# B&R Automation Studio project prac1
Automation Studio 4.12.10.39

## Configuration Config1

CPU PC_any, AutomationRuntime J4.93, Build 4.1.2, Vc V4.73.2

### Task classes (Cpu.sw)
```
Cyclic#1 (cycle 10000 us):
  Program <- Program.prg
Cyclic#4:
  Program1 <- Program1.prg
Binaries: udbdef, FWRules, TCData, sysconf, Role, User, iomap, ashwd, asfw, arconfig, ashwac
Libraries: Library
```

### Hardware
```
PC : PC_any v1.1.1.0 (OrderNumber=PC)
  ConfigurationID = prac1_Config1
  Cyclic1Duration = 10000
  Cyclic2Duration = 100000
  Cyclic3Duration = 300000
  Cyclic3Tolerance = 9900000
  FileDevice1
  FileDeviceName1 = USER
  FileDevicePath1 = USER_PATH
```

- Physical/Config1/PC/IoMap.iom: same as Physical/Config1/PC/Cpu.per
- Physical/Config1/PC/PvMap.vvm: same as Physical/Config1/PC/Cpu.per
## Logical view

Binary libraries used (declarations not repeated): operator, runtime, astime, AsIecCon

### Global.var - Global variables
```iecst
VAR
	Enable : BOOL := TRUE;
	Speed : INT;
END_VAR
```


### Program Logical/Program (ANSIC)

#### Main.c - Init, cyclic, exit code
```c
#include <bur/plctypes.h>

#ifdef _DEFAULT_INCLUDES
	#include <AsDefault.h>
#endif

void _INIT ProgramInit(void)
{
	REAL Tj = 1;
	REAL D_T = 0.01;

	fb_motor.Tm = 0.1;
	fb_motor.ke = 0.24;
	fb_motor.dt = D_T;
	fb_motor.integrator.dt = D_T;

	fb_regulator.k_p = fb_motor.ke * fb_motor.Tm / Tj;
	fb_regulator.k_i = fb_motor.ke / Tj;
	fb_regulator.dt  = D_T;
	fb_regulator.max_abs_value = 24.0;
	fb_regulator.integrator.dt = D_T;

	fb_motor_2.Tm = 0.1;
	fb_motor_2.ke = 0.24;
	fb_motor_2.dt = D_T;
	fb_motor_2.integrator.dt = D_T;

}

void _CYCLIC ProgramCyclic(void)
{

	if (Enable)
	{
		fb_regulator.e = Speed - fb_motor.w;
		FB_regulator(&fb_regulator);

		fb_motor.u = fb_regulator.u;
		FB_motor(&fb_motor);

		fb_motor_2.u = Speed * fb_motor_2.ke;
		FB_motor(&fb_motor_2);
	}
	else
	{
		fb_regulator.u = 0.0;
		fb_regulator.iyOld = 0.0;
		fb_regulator.integrator.out = 0.0;

		fb_motor.u = 0.0;
		FB_motor(&fb_motor);

		fb_motor_2.u = 0;
		FB_motor(&fb_motor_2);
	}
}
void _EXIT ProgramExit(void)
{

}
```

#### Variables.var - Local variables
```iecst
VAR
	fb_regulator : FB_regulator;
	fb_motor : FB_motor;
	fb_motor_2 : FB_motor;
END_VAR
```

### Library Logical/Library (ANSIC)

#### Library.fun - Exported functions and function blocks
```iecst
{REDUND_ERROR} FUNCTION_BLOCK FB_integrator (*TODO: Add your comment here*) (*$GROUP=User,$CAT=User,$GROUPICON=User.png,$CATICON=User.png*)
	VAR_INPUT
		out : REAL;
	END_VAR
	VAR_OUTPUT
		in : REAL;
	END_VAR
	VAR
		dt : REAL;
	END_VAR
END_FUNCTION_BLOCK

{REDUND_ERROR} {REDUND_UNREPLICABLE} FUNCTION_BLOCK FB_regulator (*TODO: Add your comment here*) (*$GROUP=User,$CAT=User,$GROUPICON=User.png,$CATICON=User.png*)
	VAR_INPUT
		e : {REDUND_UNREPLICABLE} REAL;
	END_VAR
	VAR_OUTPUT
		u : {REDUND_UNREPLICABLE} REAL;
	END_VAR
	VAR
		k_p : {REDUND_UNREPLICABLE} REAL;
		k_i : {REDUND_UNREPLICABLE} REAL;
		integrator : {REDUND_UNREPLICABLE} FB_integrator;
		iyOld : {REDUND_UNREPLICABLE} REAL;
		max_abs_value : {REDUND_UNREPLICABLE} REAL;
		dt : {REDUND_UNREPLICABLE} REAL;
	END_VAR
END_FUNCTION_BLOCK

{REDUND_ERROR} {REDUND_UNREPLICABLE} FUNCTION_BLOCK FB_motor (*TODO: Add your comment here*) (*$GROUP=User,$CAT=User,$GROUPICON=User.png,$CATICON=User.png*)
	VAR_INPUT
		u : {REDUND_UNREPLICABLE} REAL;
	END_VAR
	VAR_OUTPUT
		w : {REDUND_UNREPLICABLE} REAL;
		phi : {REDUND_UNREPLICABLE} REAL;
	END_VAR
	VAR
		integrator : {REDUND_UNREPLICABLE} FB_integrator;
		Tm : {REDUND_UNREPLICABLE} REAL;
		ke : {REDUND_UNREPLICABLE} REAL;
		dt : {REDUND_UNREPLICABLE} REAL;
	END_VAR
END_FUNCTION_BLOCK
```

#### FB_integrator.c
```c
#include <bur/plctypes.h>
#ifdef __cplusplus
	extern "C"
	{
#endif
	#include "Library.h"
#ifdef __cplusplus
	};
#endif
/* TODO: Add your comment here */
void FB_integrator(struct FB_integrator* inst)
{
	inst->out += inst->dt * inst->in;
}
```

#### FB_regulator.c
```c
#include <bur/plctypes.h>
#ifdef __cplusplus
	extern "C"
	{
#endif
	#include "Library.h"
#ifdef __cplusplus
	};
#endif
/* TODO: Add your comment here */
void FB_regulator(struct FB_regulator* inst)
{
	REAL p_channel = inst->e * inst->k_p;

	if (p_channel > inst->max_abs_value){
		p_channel = inst->max_abs_value;
	}
	if (p_channel < -inst->max_abs_value){
		p_channel = -inst->max_abs_value;
	}

	REAL i_channel = inst->k_i * inst->e - inst->iyOld;

	inst->integrator.dt = inst->dt;
	inst->integrator.in = i_channel;
	FB_integrator(&inst->integrator);
	i_channel = inst->integrator.out;

	REAL reg = p_channel + i_channel;

	inst->u = reg;
	if (reg > inst->max_abs_value){
		inst->u = inst->max_abs_value;
	}
	if (reg < -inst->max_abs_value){
		inst->u = -inst->max_abs_value;
	}

	inst->iyOld = reg - inst->u;

}
```

#### FB_motor.c
```c
#include <bur/plctypes.h>
#ifdef __cplusplus
	extern "C"
	{
#endif
	#include "Library.h"
#ifdef __cplusplus
	};
#endif
/* TODO: Add your comment here */
void FB_motor(struct FB_motor* inst)
{

	REAL e = inst->u / inst->ke - inst->w;

	inst->integrator.dt = inst->dt;
	inst->integrator.in = e / inst->Tm;
	FB_integrator(&inst->integrator);
	inst->w = inst->integrator.out;

	inst->phi = inst->phi + inst->w * inst->dt;
}
```

### Program Logical/Program1 (ANSIC)

#### Main.c - Init, cyclic, exit code
```c
#include <bur/plctypes.h>

#ifdef _DEFAULT_INCLUDES
	#include <AsDefault.h>
#endif

void _INIT ProgramInit(void)
{

}

void _CYCLIC ProgramCyclic(void)
{
	counter++;
	if (counter >= 10 && counter < 20){
		Speed = 50;
	}
	else if (counter >= 20){
		Speed = 0;
		counter = 0;
	}
}

void _EXIT ProgramExit(void)
{

}
```

#### Variables.var - Local variables
```iecst
VAR
	counter : INT := 0;
END_VAR
```
